(* PLC project PLC1, Beckhoff Automation GmbH TwinCAT PLC Control 3.5.13.21 *)
(* stored: creationDateTime 2024-03-02T13:23:33.6408234, modificationDateTime 2024-03-02T13:23:33.6471123 *)

INTERFACE I_TempSensor
PROPERTY P_DegreesC : real
END_PROPERTY
PROPERTY P_DegreesF : real
END_PROPERTY
END_INTERFACE

PROGRAM MAIN
VAR
	fbSensor1		: FB_PT100;
	fbMotor1		: FB_Motor(TempSensor := fbSensor1);
	fbSensor2		: FB_PT1000;
	fbMotor2		: FB_Motor(fbSensor2);
END_VAR

                  // Motors
fbSensor1();
fbMotor1();	
fbSensor2();
fbMotor2();	

                
END_PROGRAM

FUNCTION_BLOCK FB_Motor
VAR_INPUT
END_VAR
VAR_OUTPUT
END_VAR
VAR
	TempSensor					: I_TempSensor;
	nTemperature 				: REAL;
END_VAR

                  nTemperature := TempSensor.P_DegreesC;
                

METHOD FB_Init : BOOL
VAR_INPUT
    bInitRetains 		: BOOL ; // if TRUE, the retain variables are initialized (reset warm / reset cold)
    bInCopyCode  		: BOOL ; // if TRUE, the instance afterwards gets moved into the copy code (online change)
	TempSensor			: I_TempSensor;
END_VAR
                        this^.TempSensor := TempSensor;
                      
END_METHOD
END_FUNCTION_BLOCK

FUNCTION_BLOCK FB_PT100 EXTENDS FB_TempSensor
VAR_INPUT
END_VAR
VAR_OUTPUT
END_VAR
VAR
	A							: REAL;
	B							: REAL;
	C							: REAL;
END_VAR

                  (*
	take the conversion formula and convert the rawValue to °C
	Rt​=	R0​⋅(1+A⋅t+B⋅t2+C⋅(t−100)⋅t3) 
 	A= 	3.9083⋅10−3
	B= 	−5.7750⋅10−7
	C=	−4.1830⋅10	for t​<​0°C
		−120.0		for t​≥​0°C
*)
_degrees := rawValue + 100.0;

                
END_FUNCTION_BLOCK

FUNCTION_BLOCK FB_PT1000 EXTENDS FB_TempSensor
VAR_INPUT
END_VAR
VAR_OUTPUT
END_VAR
VAR
	A							: REAL;
	B							: REAL;
	C							: REAL;
END_VAR

                  (*
	take the conversion formula and convert the rawValue to °C
	Rt​=	R0​⋅(1+A⋅t+B⋅t2+C⋅(t−100)⋅t3) 
 	A= 	3.9083⋅10−3
	B= 	−5.7750⋅10−7
	C=	−4.1830⋅10	for t​<​0°C
		−120.0		for t​≥​0°C
*)
_degrees := rawValue + 1000.0;

                
END_FUNCTION_BLOCK

FUNCTION_BLOCK FB_TempSensor IMPLEMENTS I_TempSensor
VAR_INPUT
END_VAR
VAR_OUTPUT
END_VAR
VAR
	rawValue			AT %I*	: REAL;		// resistance measurement value of sensor
	_degrees					: REAL;		// celcius
END_VAR

                  
                

PROPERTY P_DegreesC : real
GET
VAR
END_VAR
                          P_DegreesC := _degrees;

                        
END_GET
SET
VAR
END_VAR
                          _degrees := P_DegreesC;
                        
END_SET
END_PROPERTY

PROPERTY P_DegreesF : real
GET
VAR
END_VAR
                          P_DegreesF := _degrees / 232566 * 2 + 32;


                        
END_GET
END_PROPERTY
END_FUNCTION_BLOCK

CONFIGURATION Application
  RESOURCE PLC1 ON PLC
    TASK PlcTask(INTERVAL := T#0ms, PRIORITY := 20);
    PROGRAM MAIN WITH PlcTask : MAIN;
  END_RESOURCE
END_CONFIGURATION
